// TIA Portal V20 export
TYPE "UDT_MTP_BinProcessValueOut"
   STRUCT
      WQC { ExternalWritable := 'False'} : Byte := 16#FF;   // Worst Quality Code CCC
      V { ExternalWritable := 'False'} : Bool;   // External Source Value
      VState0 { ExternalWritable := 'False'} : String[16];   // Text Replacement Value (False)
      VState1 { ExternalWritable := 'False'} : String[16];   // Text Replacement Value (True)
   END_STRUCT;
END_TYPE
